(* IEC 61131-3 sources: FeedingMachine/src/StateMachine/StateObject, 7 files *)

(* ---- ErrorState.st ---- *)
USING TankValveLib;
USING Siemens.Simatic.S71500.MotionControl;

NAMESPACE Siemens.Simatic.TCC2023.StateMachine

    CLASS PUBLIC ErrorState IMPLEMENTS IState
        VAR
            _feedAxis  : itfPosAxis;
            _tank:REF_TO Tank;
            canGoNext:BOOL:=FALSE;
        END_VAR

        //执行动作逻辑
        METHOD PUBLIC ExcuteJob
            VAR_EXTERNAL
               resetError : BOOL;
            END_VAR
            IF resetError THEN
                canGoNext:=TRUE;
                _feedAxis.ResetAlarms();
            END_IF;
        END_METHOD

        //处理状态
        METHOD PUBLIC HandleState
            VAR_INPUT
                context : REF_TO FeedingMachine;
                tank : REF_TO Tank;
                feedAxis : itfPosAxis;
            END_VAR
            VAR_EXTERNAL
                sinkEmptySensor : BOOL;
                axisStop : BOOL;
                powerOff : BOOL;
                tankEmptySensor : BOOL;
            END_VAR

            this._tank:=tank;
            this._feedAxis:=feedAxis;

            //执行Action
            this.ExcuteJob();

            //断电或空罐
            IF powerOff OR tankEmptySensor THEN
                 //切换到OFFState状态对象
                context^.SetState(context^.GetOffState(),_tank,_feedAxis);
            END_IF;

            //等待可跳转信号
            IF canGoNext THEN
                canGoNext:=FALSE;
                IF axisStop OR sinkEmptySensor THEN
                    //切换到StopState状态对象
                    context^.SetState(context^.GetStopState(),_tank,_feedAxis);
                ELSE
                //切换到Ready状态对象
                context^.SetState(context^.GetReadyState(),_tank,_feedAxis);
                END_IF;
            END_IF;
        END_METHOD

        //获取状态
        METHOD PUBLIC GetState : STRING
            GetState:='Error';
        END_METHOD

    END_CLASS

END_NAMESPACE

(* ---- FillSinkState.st ---- *)
USING TankValveLib;
USING Siemens.Simatic.S71500.MotionControl;

NAMESPACE Siemens.Simatic.TCC2023.StateMachine

    CLASS PUBLIC FillSinkState IMPLEMENTS IState
        VAR
            _feedAxis  : itfPosAxis;
            _tank:REF_TO Tank;
        END_VAR

        //执行动作逻辑
        METHOD PUBLIC ExcuteJob
            _tank^.Feeding();
        END_METHOD

        //处理状态
        METHOD PUBLIC HandleState
            VAR_INPUT
                context : REF_TO FeedingMachine;
                tank : REF_TO Tank;
                feedAxis : itfPosAxis;
            END_VAR
            VAR_EXTERNAL
                sinkFullSensor:BOOL;
                powerOff : BOOL;
                tankEmptySensor : BOOL;
            END_VAR

            this._tank:=tank;
            this._feedAxis:=feedAxis;

            //执行Action
            this.ExcuteJob();

            //断电或空罐
            IF powerOff OR tankEmptySensor THEN
                //切换到OFFState状态对象
                context^.SetState(context^.GetOffState(),_tank,_feedAxis);
            END_IF;

            //等待可跳转信号
            IF sinkFullSensor THEN
                //切换到ReadyState状态对象
                context^.SetState(context^.GetReadyState(),_tank,_feedAxis);
            END_IF;
        END_METHOD

        //获取状态
        METHOD PUBLIC GetState : STRING
            GetState:='fillingSink';
        END_METHOD

    END_CLASS

END_NAMESPACE

(* ---- FillTankState.st ---- *)
USING TankValveLib;
USING Siemens.Simatic.S71500.MotionControl;

NAMESPACE Siemens.Simatic.TCC2023.StateMachine

    CLASS PUBLIC FillTankState IMPLEMENTS IState
        VAR
            _feedAxis  : itfPosAxis;
            _tank:REF_TO Tank;
        END_VAR

        //执行动作逻辑
        METHOD Public ExcuteJob
            _tank^.Filling();
            _feedAxis.PowerOff();
        END_METHOD

        //处理状态
        METHOD PUBLIC HandleState
            VAR_INPUT
                context:REF_TO FeedingMachine;
                tank:REF_TO Tank;
                feedAxis:itfPosAxis;
            END_VAR
            VAR_EXTERNAL
                tankFullSensor :BOOL;
                powerOff : BOOL;
                tankEmptySensor : BOOL;
            END_VAR

            this._tank:=tank;
            this._feedAxis:=feedAxis;

            //执行Action
            this.ExcuteJob();

            //断电或空罐
            IF powerOff OR tankEmptySensor THEN
                //切换到OFFState状态对象
                context^.SetState(context^.GetOffState(),_tank,_feedAxis);

            END_IF;
            //等待可跳转信号
            IF tankFullSensor THEN
                //切换到fILLSinkState状态对象
                context^.SetState(context^.GetFillSinkState(),_tank,_feedAxis);
            END_IF;
        END_METHOD

        //获取状态
        METHOD PUBLIC GetState : STRING
            GetState:='Filling Tank';
        END_METHOD

    END_CLASS

END_NAMESPACE

(* ---- OffState.st ---- *)
USING TankValveLib;
USING Siemens.Simatic.S71500.MotionControl;

NAMESPACE Siemens.Simatic.TCC2023.StateMachine

    CLASS PUBLIC OffState IMPLEMENTS IState
        VAR
            _feedAxis  : itfPosAxis;
            _tank: REF_TO Tank;
        END_VAR

        //执行动作逻辑
        METHOD PUBLIC ExcuteJob
            _tank^.Close();
            _feedAxis.PowerOff();
        END_METHOD

        //处理状态
        METHOD PUBLIC HandleState
            VAR_INPUT
                context : REF_TO FeedingMachine;
                tank : REF_TO Tank;
                feedAxis : itfPosAxis;
            END_VAR
            VAR_EXTERNAL
                powerOn :BOOL;
                powerOff : BOOL;
            END_VAR

            this._tank:=tank;
            this._feedAxis:=feedAxis;

            //执行Action
            this.ExcuteJob();

            //等待可跳转信号
            IF powerOn AND NOT(powerOff) THEN
                //切换到FillSink状态对象
                context^.SetState(context^.GetFillTankState(),_tank,_feedAxis);
            END_IF;
        END_METHOD

        //获取状态
        METHOD PUBLIC GetState : STRING
            GetState:='OFF';
        END_METHOD

    END_CLASS

END_NAMESPACE

(* ---- ReadyState.st ---- *)
USING TankValveLib;
USING Siemens.Simatic.S71500.MotionControl;

NAMESPACE Siemens.Simatic.TCC2023.StateMachine

    CLASS PUBLIC ReadyState IMPLEMENTS IState
        VAR
            _feedAxis  : itfPosAxis;
            _tank:REF_TO Tank;
            canGoNext:BOOL:=FALSE;
        END_VAR

        //执行动作逻辑
        METHOD PUBLIC ExcuteJob
            VAR_EXTERNAL
                axisStart:BOOL;
                errorID : WORD;
            END_VAR
            VAR
                AxHomeCmd:itfCommand;
            END_VAR
            _tank^.Close();
            IF axisStart THEN
                _feedAxis.PowerOn();
                AxHomeCmd:=_feedAxis.HomeDirect(Position:=LREAL#0.0, Mode:=HomingModeDirect#ActualPositionAbsolute);
                IF AxHomeCmd.Error() THEN
                    errorID:=Word#16#8003;
                ELSE
                    canGoNext:=TRUE;
                END_IF;
            END_IF;
        END_METHOD

        //处理状态
        METHOD PUBLIC HandleState
            VAR_INPUT
                context : REF_TO FeedingMachine;
                tank : REF_TO Tank;
                feedAxis : itfPosAxis;
            END_VAR
            VAR_EXTERNAL
                powerOff : BOOL;
                tankEmptySensor : BOOL;
                errorID : WORD;
                sinkEmptySensor:Bool;
            END_VAR

            this._tank:=tank;
            this._feedAxis:=feedAxis;

            //执行Action
            this.ExcuteJob();

            //轴控错误
            IF ErrorID <> Word#16#0000 THEN
                //切换到Error状态对象
                context^.SetState(context^.GetErrorState(),_tank,_feedAxis);;
            END_IF;

            //断电或空罐
            IF powerOff OR tankEmptySensor THEN
                 //切换到OFFState状态对象
                context^.SetState(context^.GetOffState(),_tank,_feedAxis);
            END_IF;

            //等待可跳转信号
            IF canGoNext AND NOT(sinkEmptySensor) THEN
                canGoNext:=FALSE;
                //切换到RunState状态对象
                context^.SetState(context^.GetRunState(),_tank,_feedAxis);
            END_IF;
        END_METHOD

        //获取状态
        METHOD PUBLIC GetState : STRING
            GetState:='Ready';
        END_METHOD

    END_CLASS

END_NAMESPACE

(* ---- RunState.st ---- *)
USING TankValveLib;
USING Siemens.Simatic.S71500.MotionControl;

NAMESPACE Siemens.Simatic.TCC2023.StateMachine

    CLASS PUBLIC RunState IMPLEMENTS IState
        VAR
            _feedAxis  : itfPosAxis;
            _tank: REF_TO Tank;
        END_VAR

        //执行动作逻辑
        METHOD PUBLIC ExcuteJob
            VAR
                AxMoveCmd:itfCommand;
            END_VAR
            VAR_EXTERNAL
                errorID : WORD;
            END_VAR
            AxMoveCmd:=_feedAxis.MoveAbsolute(Position:=LREAL#10000.0, Velocity := LREAL#50.0, Direction := DirectionModulo#ShortestDistance);
            IF AxMoveCmd.Error() THEN
              errorID:=Word#16#8004;
            END_IF;
        END_METHOD

        //处理状态
        METHOD PUBLIC HandleState
            VAR_INPUT
                context : REF_TO FeedingMachine;
                tank : REF_TO Tank;
                feedAxis : itfPosAxis;
            END_VAR
            VAR_EXTERNAL
                axisStop:BOOL;
                sinkEmptySensor : BOOL;
                powerOff : BOOL;
                tankEmptySensor : BOOL;
                errorID : WORD;
            END_VAR

            this._tank:=tank;
            this._feedAxis:=feedAxis;

            //执行Action
            this.ExcuteJob();

            //轴控错误
            IF ErrorID <> Word#16#0000 THEN
                //切换到Error状态对象
                context^.SetState(context^.GetErrorState(),_tank,_feedAxis);;
            END_IF;

            //断电或空罐
            IF powerOff OR tankEmptySensor THEN
                 //切换到OFFState状态对象
                context^.SetState(context^.GetOffState(),_tank,_feedAxis);
            END_IF;

            //等待可跳转信号
            IF axisStop OR sinkEmptySensor THEN
                //切换到StopState状态对象
                context^.SetState(context^.GetStopState(),_tank,_feedAxis);
            END_if;
        END_METHOD

        //获取状态
        METHOD PUBLIC GetState : STRING
            GetState:='Runing';
        END_METHOD

    END_CLASS

END_NAMESPACE

(* ---- StopState.st ---- *)
USING TankValveLib;
USING Siemens.Simatic.S71500.MotionControl;

NAMESPACE Siemens.Simatic.TCC2023.StateMachine

    CLASS PUBLIC StopState IMPLEMENTS IState
        VAR
            _feedAxis  : itfPosAxis;
            _tank:REF_TO Tank;
        END_VAR

        //执行动作逻辑
        METHOD PUBLIC ExcuteJob
            VAR
                AxHaltCmd:itfCommand;
            END_VAR
            VAR_EXTERNAL
                errorID : WORD;
            END_VAR

            AxHaltCmd:=_feedAxis.Halt();

            IF AxHaltCmd.Error() THEN
                errorID:=Word#16#8005;
            END_IF;
        END_METHOD

        //处理状态
        METHOD PUBLIC HandleState
            VAR_INPUT
                context : REF_TO FeedingMachine;
                tank : REF_TO Tank;
                feedAxis : itfPosAxis;
            END_VAR
            VAR_EXTERNAL
                axisStart : BOOL;
                axisStop : BOOL;
                powerOff : BOOL;
                tankEmptySensor : BOOL;
                errorID : WORD;
            END_VAR
            this._tank:=tank;
            this._feedAxis:=feedAxis;

            //执行Action
            this.ExcuteJob();

             //轴控错误
             IF ErrorID <> Word#16#0000 THEN
                //切换到Error状态对象
                context^.SetState(context^.GetErrorState(),_tank,_feedAxis);;
            END_IF;

            //断电或空罐
            IF powerOff OR tankEmptySensor THEN
                 //切换到OFFState状态对象
                context^.SetState(context^.GetOffState(),_tank,_feedAxis);
                END_IF;

            //等待可跳转信号
            IF axisStart AND NOT axisStop THEN
                //切换到FillSinkState状态对象
                context^.SetState(context^.GetFillSinkState(),_tank,_feedAxis);
            END_IF;

        END_METHOD

        //获取状态
        METHOD PUBLIC GetState : STRING
            GetState:='Stoped';
        END_METHOD

    END_CLASS

END_NAMESPACE
